ABB RAPID module: RNL__ModuleExample.modx

MODULE RNL__ModuleExample

    PERS dataType dataType_ModuleExample:="ModuleExample";
    PERS dataPointer ModuleExample:=["ModuleExample","ModuleExample",0,"","",0,""];


    LOCAL PROC config()
    ENDPROC

    LOCAL PROC init()
    ENDPROC

    LOCAL PROC update()
    ENDPROC

ENDMODULE
